# EPICS substitutions: smargonBuilder/iocs/BL99I-LCH-IOC-01/BL99I-LCH-IOC-01App/Db/BL99I-LCH-IOC-01_expanded.substitutions
# This file was automatically generated on Thu 06 Sep 2018 11:58:55 BST from
# source: /home/jjc62351/work/Builder/smargonBuilder/etc/makeIocs/BL99I-LCH-IOC-01.xml
#
# *** Please do not edit this file: edit the source file instead. ***
#

file $(AUTOSAVE)/db/dlssrfile.template
{
pattern { device, file }
    { "BL03I-MO-IOC-06", "0" }
    { "BL03I-MO-IOC-06", "1" }
    { "BL03I-MO-IOC-06", "2" }
}

file $(AUTOSAVE)/db/dlssrstatus.template
{
pattern { device, name }
    { "BL03I-MO-IOC-06", "BL03I-MO-IOC-06.AUTOSAVE" }
}

# Macros:
#  IOC  Device prefix
file $(DEVIOCSTATS)/db/iocAdminSoft.db
{
pattern { IOC }
    { "BL03I-MO-IOC-06" }
}

# Macros:
#  IOC  Device prefix
file $(DEVIOCSTATS)/db/iocAdminScanMon.db
{
pattern { IOC }
    { "BL03I-MO-IOC-06" }
}

# Macros:
#  name      name for gui elements
#  EDM_FILE  edm screen, defaults to ioc_stats_softdls.edl
#  IOC       ioc name
file $(DEVIOCSTATS)/db/iocGui.db
{
pattern { name, EDM_FILE, IOC }
    { "MO6", "ioc_stats_softdls.edl", "BL03I-MO-IOC-06" }
}

# Macros:
#  PORT      The asyn port for the pmac controller
#  P         PV Prefix
#  NAXES     Number of axes
#  TIMEOUT   Timeout for controller communication
#  FEEDRATE  feedrate below which we go into error
#  CSG0      Name for Coordinate System Group 0
#  CSG1      Name for Coordinate System Group 1
#  CSG2      Name for Coordinate System Group 2
#  CSG3      Name for Coordinate System Group 3
#  CSG4      Name for Coordinate System Group 4
#  CSG5      Name for Coordinate System Group 5
#  CSG6      Name for Coordinate System Group 6
#  CSG7      Name for Coordinate System Group 7
file $(PMAC)/db/pmacController.template
{
pattern { PORT, P, NAXES, TIMEOUT, FEEDRATE, CSG0, CSG1, CSG2, CSG3, CSG4, CSG5, CSG6, CSG7 }
    { "PPMAC1", "BL03I-MO-SGON-01", "8", "4", "100", "", "", "", "", "", "", "", "" }
    { "BRICK5", "BL03I-MO-STEP-05", "8", "4", "100", "", "", "", "", "", "", "", "" }
}

# Macros:
#  DEVICE    Pmac/Geobrick name
#  PLC       PLC for CPU load monitoring, e.g. 5
#  NAXES     Number of axes
#  PORT      Delta tau motor controller
#  name      Object and gui association name
#  FEEDRATE  feedrate below which we go into error
#  TIMEOUT   timeout for brick communications
file $(PMAC)/db/powerPmacStatus.template
{
pattern { DEVICE, PLC, NAXES, PORT, name, FEEDRATE, TIMEOUT }
    { "BL03I-MO-PPMAC-01", "13", "8", "PPMAC1", "PPMAC_STATUS", "0", "100" }
}

# Macros:
#  PMAC  Pmac/Geobrick name
#  AXIS  Axis number
#  PORT  Asyn port
file $(PMAC)/db/pmacStatusAxis.template
{
pattern { PMAC, AXIS, PORT }
    { "BL03I-MO-PPMAC-01", "1", "PPMAC1" }
    { "BL03I-MO-PPMAC-01", "2", "PPMAC1" }
    { "BL03I-MO-PPMAC-01", "3", "PPMAC1" }
    { "BL03I-MO-PPMAC-01", "4", "PPMAC1" }
    { "BL03I-MO-PPMAC-01", "5", "PPMAC1" }
    { "BL03I-MO-PPMAC-01", "6", "PPMAC1" }
    { "BL03I-MO-PPMAC-01", "7", "PPMAC1" }
    { "BL03I-MO-PPMAC-01", "8", "PPMAC1" }
    { "BL03I-MO-STEP-05", "1", "BRICK5" }
    { "BL03I-MO-STEP-05", "2", "BRICK5" }
    { "BL03I-MO-STEP-05", "3", "BRICK5" }
    { "BL03I-MO-STEP-05", "4", "BRICK5" }
    { "BL03I-MO-STEP-05", "5", "BRICK5" }
    { "BL03I-MO-STEP-05", "6", "BRICK5" }
    { "BL03I-MO-STEP-05", "7", "BRICK5" }
    { "BL03I-MO-STEP-05", "8", "BRICK5" }
}

# Macros:
#  P                Device Prefix
#  M                Device Suffix
#  PORT             Delta tau motor controller
#  ADDR             Address on controller
#  DESC             Description, displayed on EDM screen
#  MRES             Motor Step Size (EGU)
#  VELO             Velocity (EGU/s)
#  PREC             Display Precision
#  EGU              Engineering Units
#  TWV              Tweak Step Size (EGU)
#  DTYP             DTYP of record
#  DIR              User Direction
#  VBAS             Base Velocity (EGU/s)
#  VMAX             Max Velocity (EGU/s), defaults to VELO
#  ACCL             Seconds to Velocity
#  BDST             BL Distance (EGU)
#  BVEL             BL Velocity (EGU/s)
#  BACC             BL Seconds to Veloc.
#  DHLM             Dial High Limit
#  DLLM             Dial Low Limit
#  HLM              User High Limit
#  LLM              User Low Limit
#  HLSV             HW Lim. Violation Svr
#  INIT             Startup commands
#  SREV             Steps per Revolution
#  RRES             Readback Step Size (EGU)
#  ERES             Encoder Step Size (EGU)
#  JAR              Jog Acceleration (EGU/s^2)
#  UEIP             Use Encoder If Present
#  URIP             Use RDBL If Present
#  RDBL             Readback Location, set URIP = 1 if you specify this
#  RLNK             Readback output link
#  RTRY             Max retry count
#  DLY              Readback settle time (s)
#  OFF              User Offset (EGU)
#  RDBD             Retry Deadband (EGU)
#  FOFF             Freeze Offset, 0=variable, 1=frozen
#  ADEL             Alarm monitor deadband (EGU)
#  NTM              New Target Monitor, only set to 0 for soft motors
#  FEHIGH           HIGH limit for following error
#  FEHIHI           HIHI limit for following error
#  FEHHSV           HIHI alarm severity for following error
#  FEHSV            HIGH alarm severity for following error
#  SCALE            Scale factor, if pmacSetAxisScale is used this should be set
#  HOMEVIS          If 1 then home is visible on the gui
#  HOMEVISSTR       If HOMEVIS=0, then display this text on the gui instead
#  name             Object name and gui association name
#  alh              Set this to alh to add the motor to the alarm handler and send emails,
#  gda_name         Name to export this as to GDA
#  gda_desc         Description to export this as to GDA
#  SPORT            Delta tau motor controller comms port
#  HOME             Prefix for autohome instance. Defaults to $(P). If unspecified,
#  ALLOW_HOMED_SET  Set to a blank to allow this axis to have its homed
file $(PMAC)/db/dls_pmac_asyn_motor.template
{
pattern { P, M, PORT, ADDR, DESC, MRES, VELO, PREC, EGU, TWV, DTYP, DIR, VBAS, VMAX, ACCL, BDST, BVEL, BACC, DHLM, DLLM, HLM, LLM, HLSV, INIT, SREV, RRES, ERES, JAR, UEIP, URIP, RDBL, RLNK, RTRY, DLY, OFF, RDBD, FOFF, ADEL, NTM, FEHIGH, FEHIHI, FEHHSV, FEHSV, SCALE, HOMEVIS, HOMEVISSTR, name, alh, gda_name, gda_desc, SPORT, HOME, PMAC, ALLOW_HOMED_SET }
    { "BL03I-MO-SGON-01", ":MOTOR_1", "PPMAC1", "1", "SmarGon Y", ".000005", "5", "5", "mm", "1", "asynMotor", "0", "0", "$(VELO)", "0.10", "0", "0", "", "0", "0", "", "", "NO_ALARM", "", "200", "", "", "", "0", "0", "", "", "0", "0", "0", "", "0", "0", "1", "0", "0", "NO_ALARM", "NO_ALARM", "200", "0", "Use Home Button", "", "None", "", "$(DESC)", "SSHP", "$(P)", "BL03I-MO-SGON-01", "#" }
    { "BL03I-MO-SGON-01", ":MOTOR_2", "PPMAC1", "2", "SmarGon Z", ".000005", "5", "5", "mm", "1", "asynMotor", "0", "0", "$(VELO)", "0.10", "0", "0", "", "0", "0", "", "", "NO_ALARM", "", "200", "", "", "", "0", "0", "", "", "0", "0", "0", "", "0", "0", "1", "0", "0", "NO_ALARM", "NO_ALARM", "200", "0", "Use Home Button", "", "None", "", "$(DESC)", "SSHP", "$(P)", "BL03I-MO-SGON-01", "#" }
    { "BL03I-MO-SGON-01", ":MOTOR_3", "PPMAC1", "3", "SmarGon X1", ".000005", "5", "5", "mm", "1", "asynMotor", "0", "0", "$(VELO)", "0.10", "0", "0", "", "0", "0", "", "", "NO_ALARM", "", "200", "", "", "", "0", "0", "", "", "0", "0", "0", "", "0", "0", "1", "0", "0", "NO_ALARM", "NO_ALARM", "200", "0", "Use Home Button", "", "None", "", "$(DESC)", "SSHP", "$(P)", "BL03I-MO-SGON-01", "#" }
    { "BL03I-MO-SGON-01", ":MOTOR_4", "PPMAC1", "4", "SmarGon X2", ".000005", "5", "5", "mm", "1", "asynMotor", "0", "0", "$(VELO)", "0.10", "0", "0", "", "0", "0", "", "", "NO_ALARM", "", "200", "", "", "", "0", "0", "", "", "0", "0", "0", "", "0", "0", "1", "0", "0", "NO_ALARM", "NO_ALARM", "200", "0", "Use Home Button", "", "None", "", "$(DESC)", "SSHP", "$(P)", "BL03I-MO-SGON-01", "#" }
    { "BL03I-MO-SGON-01", ":MOTOR_5", "PPMAC1", "5", "SmarGon Phi", ".000005", "60", "5", "deg", "1", "asynMotor", "0", "0", "$(VELO)", "0.10", "0", "0", "", "0", "0", "", "", "NO_ALARM", "", "200", "", "", "", "0", "0", "", "", "0", "0", "0", "", "0", "0", "1", "0", "0", "NO_ALARM", "NO_ALARM", "200", "0", "Use Home Button", "", "None", "", "$(DESC)", "SSHP", "$(P)", "BL03I-MO-SGON-01", "#" }
    { "BL03I-MO-SGON-01", ":MOTOR_6", "PPMAC1", "6", "SmarGon Omega", ".000005", "180", "5", "deg", "1", "asynMotor", "0", "0", "$(VELO)", "0.10", "0", "0", "", "0", "0", "", "", "NO_ALARM", "", "200", "", "", "", "0", "0", "", "", "0", "0", "0", "", "0", "0", "1", "0", "0", "NO_ALARM", "NO_ALARM", "200", "0", "Use Home Button", "", "None", "", "$(DESC)", "SSHP", "$(P)", "BL03I-MO-SGON-01", "#" }
    { "BL03I-MO-GONIO-01", ":X", "BRICK5", "1", "Gonio Positioner X", "0.00005", "12", "5", "mm", "1", "asynMotor", "0", "0", "$(VELO)", "0.1", "0", "0", "", "150", "-50", "", "", "MAJOR", "", "1000", "", "", "", "0", "0", "", "", "0", "0", "0", "", "0", "0", "1", "0", "0", "NO_ALARM", "NO_ALARM", "1", "1", "Use motor summary screen", "GONP.X", "None", "", "$(DESC)", "BRICK5port", "$(P)", "BL03I-MO-STEP-05", "#" }
    { "BL03I-MO-GONIO-01", ":Y", "BRICK5", "2", "Gonio Positioner Y", "0.00005", "9", "5", "mm", "1", "asynMotor", "0", "0", "$(VELO)", "0.1", "0", "0", "", "12", "-10", "", "", "MAJOR", "", "1000", "", "", "", "0", "0", "", "", "0", "0", "0", "", "0", "0", "1", "0", "0", "NO_ALARM", "NO_ALARM", "1", "1", "Use motor summary screen", "GONP.Y", "None", "", "$(DESC)", "BRICK5port", "$(P)", "BL03I-MO-STEP-05", "#" }
    { "BL03I-MO-GONIO-01", ":Z", "BRICK5", "3", "Gonio Positioner Z", "0.00005", "12", "5", "mm", "1", "asynMotor", "0", "0", "$(VELO)", "0.1", "0", "0", "", "25", "-25", "", "", "MAJOR", "", "1000", "", "", "", "0", "0", "", "", "0", "0", "0", "", "0", "0", "1", "0", "0", "NO_ALARM", "NO_ALARM", "1", "1", "Use motor summary screen", "GONP.Z", "None", "", "$(DESC)", "BRICK5port", "$(P)", "BL03I-MO-STEP-05", "#" }
    { "BL03I-MO-GONIO-01", ":OMEGA", "BRICK5", "7", "Gonio Omega", "0.000015203", "45", "5", "deg", "1", "asynMotor", "0", "0", "$(VELO)", "0.1", "0", "0", "", "", "", "", "", "MAJOR", "", "1000", "", "", "", "0", "0", "", "", "0", "0", "0", "", "0", "0", "1", "0", "0", "NO_ALARM", "NO_ALARM", "1", "1", "Use motor summary screen", "GONIO.OMEGA", "None", "", "$(DESC)", "BRICK5port", "$(P)", "BL03I-MO-STEP-05", "#" }
    { "BL03I-MO-GONIO-01", ":PLATEY", "BRICK5", "5", "Plate Centering Y", "0.0001", "5", "5", "mm", "1", "asynMotor", "0", "0", "$(VELO)", "0.2", "0", "0", "", "66.15", "-33.85", "", "", "MAJOR", "", "1000", "", "", "", "0", "0", "", "", "0", "0", "-16.15", "", "0", "0", "1", "0", "0", "NO_ALARM", "NO_ALARM", "1", "1", "Use motor summary screen", "GONIO.PLATEY", "None", "", "$(DESC)", "BRICK5port", "$(P)", "BL03I-MO-STEP-05", "#" }
    { "BL03I-MO-GONIO-01", ":PLATEZ", "BRICK5", "6", "Plate Centering Z", "0.0001", "5", "5", "mm", "1", "asynMotor", "0", "0", "$(VELO)", "0.2", "0", "0", "", "12.5", "-12.5", "", "", "MAJOR", "", "1000", "", "", "", "0", "0", "", "", "0", "0", "-0.5", "", "0", "0", "1", "0", "0", "NO_ALARM", "NO_ALARM", "1", "1", "Use motor summary screen", "GONIO.PLATEZ", "None", "", "$(DESC)", "BRICK5port", "$(P)", "BL03I-MO-STEP-05", "#" }
}

# Macros:
#  PORT     The asyn port for the pmac cs controller
#  PMAC     PV Prefix for the motor controller
#  CS       Coordinate System Number for the cs controller
#  TIMEOUT  Timeout for controller communication
file $(PMAC)/db/pmacCsController.template
{
pattern { PORT, PMAC, CS, TIMEOUT }
    { "CS1", "BL03I-MO-SGON-01", "1", "4" }
}

# Macros:
#  P           Device Prefix
#  M           Device Suffix
#  PORT        Delta tau motor controller
#  ADDR        Address on controller
#  DESC        Description, displayed on EDM screen
#  MRES        Motor Step Size (EGU)
#  VELO        Velocity (EGU/s)
#  PREC        Display Precision
#  EGU         Engineering Units
#  TWV         Tweak Step Size (EGU)
#  DTYP        DTYP of record
#  DIR         User Direction
#  VBAS        Base Velocity (EGU/s)
#  VMAX        Max Velocity (EGU/s), defaults to VELO
#  ACCL        Seconds to Velocity
#  BDST        BL Distance (EGU)
#  BVEL        BL Velocity (EGU/s)
#  BACC        BL Seconds to Veloc.
#  DHLM        Dial High Limit
#  DLLM        Dial Low Limit
#  HLM         User High Limit
#  LLM         User Low Limit
#  HLSV        HW Lim. Violation Svr
#  INIT        Startup commands
#  SREV        Steps per Revolution
#  RRES        Readback Step Size (EGU)
#  ERES        Encoder Step Size (EGU)
#  JAR         Jog Acceleration (EGU/s^2)
#  UEIP        Use Encoder If Present
#  URIP        Use RDBL If Present
#  RDBL        Readback Location, set URIP = 1 if you specify this
#  RLNK        Readback output link
#  RTRY        Max retry count
#  DLY         Readback settle time (s)
#  OFF         User Offset (EGU)
#  RDBD        Retry Deadband (EGU)
#  FOFF        Freeze Offset, 0=variable, 1=frozen
#  ADEL        Alarm monitor deadband (EGU)
#  NTM         New Target Monitor, only set to 0 for soft motors
#  FEHIGH      HIGH limit for following error
#  FEHIHI      HIHI limit for following error
#  FEHHSV      HIHI alarm severity for following error
#  FEHSV       HIGH alarm severity for following error
#  SCALE       Scale factor, if pmacSetAxisScale is used this should be set
#  HOMEVIS     If 1 then home is visible on the gui
#  HOMEVISSTR  If HOMEVIS=0, then display this text on the gui instead
#  name        Object name and gui association name
#  alh         Set this to alh to add the motor to the alarm handler and send emails,
#  gda_name    Name to export this as to GDA
#  gda_desc    Description to export this as to GDA
file $(PMAC)/db/dls_pmac_cs_asyn_motor.template
{
pattern { P, M, PORT, ADDR, DESC, MRES, VELO, PREC, EGU, TWV, DTYP, DIR, VBAS, VMAX, ACCL, BDST, BVEL, BACC, DHLM, DLLM, HLM, LLM, HLSV, INIT, SREV, RRES, ERES, JAR, UEIP, URIP, RDBL, RLNK, RTRY, DLY, OFF, RDBD, FOFF, ADEL, NTM, FEHIGH, FEHIHI, FEHHSV, FEHSV, SCALE, HOMEVIS, HOMEVISSTR, name, alh, gda_name, gda_desc, PMAC, CS }
    { "BL03I-MO-SGON-01", ":X", "CS1", "7", "X Translation", "0.0000001", "10", "5", "mm", "1", "asynMotor", "0", "0", "$(VELO)", "0.5", "0", "0", "", "", "", "0", "0", "NO_ALARM", "", "200", "", "", "1", "0", "0", "", "", "0", "0", "0", "", "0", "0", "1", "0", "0", "NO_ALARM", "NO_ALARM", "1", "0", "Use Home Button", "SGON-X", "None", "", "$(DESC)", "BL03I-MO-SGON-01", "1" }
    { "BL03I-MO-SGON-01", ":Y", "CS1", "8", "Y Translation", "0.0000001", "10", "5", "mm", "1", "asynMotor", "0", "0", "$(VELO)", "0.5", "0", "0", "", "", "", "0", "0", "NO_ALARM", "", "200", "", "", "1", "0", "0", "", "", "0", "0", "0", "", "0", "0", "1", "0", "0", "NO_ALARM", "NO_ALARM", "1", "0", "Use Home Button", "SGON-Y", "None", "", "$(DESC)", "BL03I-MO-SGON-01", "1" }
    { "BL03I-MO-SGON-01", ":Z", "CS1", "9", "Z Translation", "0.0000001", "10", "5", "mm", "1", "asynMotor", "0", "0", "$(VELO)", "0.5", "0", "0", "", "", "", "0", "0", "NO_ALARM", "", "200", "", "", "1", "0", "0", "", "", "0", "0", "0", "", "0", "0", "1", "0", "0", "NO_ALARM", "NO_ALARM", "1", "0", "Use Home Button", "SGON-Z", "None", "", "$(DESC)", "BL03I-MO-SGON-01", "1" }
    { "BL03I-MO-SGON-01", ":OMEGA", "CS1", "1", "Omega", "0.001000", "180", "5", "deg", "1", "asynMotor", "0", "0", "$(VELO)", "0.5", "0", "0", "", "", "", "0", "0", "NO_ALARM", "", "200", "", "", "1", "0", "0", "", "", "0", "0", "0", "", "0", "0", "1", "0", "0", "NO_ALARM", "NO_ALARM", "1", "0", "Use Home Button", "SGON-OMEGA", "None", "", "$(DESC)", "BL03I-MO-SGON-01", "1" }
    { "BL03I-MO-SGON-01", ":PHI", "CS1", "2", "Phi", "0.001000", "80", "5", "deg", "1", "asynMotor", "0", "0", "$(VELO)", "0.5", "0", "0", "", "", "", "0", "0", "NO_ALARM", "", "200", "", "", "1", "0", "0", "", "", "0", "0", "0", "", "0", "0", "1", "0", "0", "NO_ALARM", "NO_ALARM", "1", "0", "Use Home Button", "SGON-PHI", "None", "", "$(DESC)", "BL03I-MO-SGON-01", "1" }
    { "BL03I-MO-SGON-01", ":CHI", "CS1", "3", "Chi", "0.0000001", "12", "5", "deg", "1", "asynMotor", "0", "0", "$(VELO)", "0.5", "1", "12", "0.5", "", "", "0", "0", "NO_ALARM", "", "200", "", "", "1", "0", "0", "", "", "0", "0", "0", "", "0", "0", "1", "0", "0", "NO_ALARM", "NO_ALARM", "1", "0", "Use Home Button", "SGON-CHI", "None", "", "$(DESC)", "BL03I-MO-SGON-01", "1" }
}

file $(BL03I)/db/Flu_Det_Protection.template
{
    { _ }
}

# Macros:
#  P           Pv Prefix
#  PLC         PLC number
#  PORT        Delta tau motor controller port
#  GRP1        Homing group 1 description
#  GRP2        Homing group 2 description
#  GRP3        Homing group 3 description
#  GRP4        Homing group 4 description
#  GRP5        Homing group 5 description
#  GRP6        Homing group 6 description
#  GRP7        Homing group 7 description
#  GRP8        Homing group 8 description
#  GRP9        Homing group 9 description
#  GRP10       Homing group 10 description
#  STATE11     Homing state 11 description
#  STATE12     Homing state 12 description
#  STATE13     Homing state 13 description
#  STATE14     Homing state 14 description
#  STATE15     Homing state 15 description
#  STATUS11    Homing status 11 description (e.g. for custom limit checks)
#  STATUS12    Homing status 12 description (e.g. for custom limit checks)
#  STATUS13    Homing status 13 description (e.g. for custom limit checks)
#  STATUS14    Homing status 14 description (e.g. for custom limit checks)
#  STATUS15    Homing status 15 description (e.g. for custom limit checks)
#  STATUSSV11  Homing status 11 severity
#  STATUSSV12  Homing status 12 severity
#  STATUSSV13  Homing status 13 severity
#  STATUSSV14  Homing status 14 severity
#  STATUSSV15  Homing status 15 severity
#  name        Object name and gui association name
#  DESC        Description
file $(PMAC)/db/autohome.template
{
pattern { P, PLC, PORT, CTRL, GRP1, GRP2, GRP3, GRP4, GRP5, GRP6, GRP7, GRP8, GRP9, GRP10, STATE11, STATE12, STATE13, STATE14, STATE15, STATUS11, STATUS12, STATUS13, STATUS14, STATUS15, STATUSSV11, STATUSSV12, STATUSSV13, STATUSSV14, STATUSSV15, name, DESC }
    { "BL03I-MO-GONIO-01", "12", "BRICK5", "BL03I-MO-STEP-05", "All", "X Translation", "Y Translation", "Z Translation", "Omega", "", "", "", "", "", "", "", "", "", "", "", "", "", "", "", "NO_ALARM", "NO_ALARM", "NO_ALARM", "NO_ALARM", "NO_ALARM", "GONP", "" }
    { "BL03I-MO-GONIO-01:PLATE", "13", "BRICK5", "BL03I-MO-STEP-05", "All", "Y Translation", "Z Translation", "", "", "", "", "", "", "", "", "", "", "", "", "", "", "", "", "", "NO_ALARM", "NO_ALARM", "NO_ALARM", "NO_ALARM", "NO_ALARM", "PLATE", "" }
}

# Macros:
#  P     Template argument
#  R     Template argument
#  PORT  Template argument
#  ADDR  Template argument
#  OMAX  Template argument
#  IMAX  Template argument
file $(ASYN)/db/asynRecord.db
{
pattern { P, R, PORT, ADDR, OMAX, IMAX }
    { "BL03I-MO-IOC-06", ":ASYN5", "BRICK5port", "0", "80", "80" }
}
